# EPICS autosave request: stdApp/Db/pid_control_settings.req
# FILE... pid_control_settings.req
# USAGE.. pid_control.db fields autosave'd.
$(P)$(PID).INP
$(P)$(PID).OUTL
$(P)$(PID).VAL
$(P)$(PID).SCAN
$(P)$(PID).HOPR
$(P)$(PID).LOPR
$(P)$(PID).DRVL
$(P)$(PID).DRVH
$(P)$(PID).FMOD
$(P)$(PID).KP
$(P)$(PID).KI
$(P)$(PID).KD
$(P)$(PID).DT
